FUNCTION Convert_DWORD_TO_DINT : Hresult
VAR_INPUT
	in : DWORD;
	out : REFERENCE TO DINT;
END_VAR
VAR
	converted : DINT;
END_VAR
VAR CONSTANT
	INCOMPATIBLE : HRESULT := 16#9811070E;
END_VAR

converted := DWORD_TO_DINT(in);

IF (DINT_TO_DWORD(converted) <> in) THEN
	Convert_DWORD_TO_DINT := INCOMPATIBLE;
	RETURN;
END_IF

out := converted;

END_FUNCTION

(* stored: Version 1.1.0.1, ProductVersion 3.1.4024.12
   POU Convert_DWORD_TO_DINT: Id {c7d62349-161f-4dd7-8590-a4f456236711}, SpecialFunc None *)
